FUNCTION_BLOCK ForceLimiterFSM IMPLEMENTS i_actionHandler
VAR_INPUT
	xEnable				: BOOL;				// Enable inputs and FSM operation
	MaxSnub				: LREAL; 			// Max Sbub (in negative lbs)
	MaxPull				: LREAL;			// Max Pull (lbs)
	Rih					: BOOL;				// Run in hole
	Pooh				: BOOL;				// Pull out of hole
	CriticalWeightRih	: LREAL;			// RIH critical weight (Cerburus Catastrophic Buckling, in negative lbs)
	CriticalWeightPooh	: LREAL;			// POOH critical weight ( Cerburus 80% pipe yield force, lbs)	
	SurpassTimeout 		: TIME  := T#10S;	// Limit surpass timeout value input
	SurpassThreshhold	: LREAL := 3.0;		// Limit surpass threshhod in %	
	CerberusDataLoaded 	: BOOL;				// Cerberus data loaded
	SurfaceWeight		: LREAL;			// Actual surface weight (lbs)	
END_VAR
VAR_OUTPUT
	Warn		: BOOL;	// Approaching limits warn
	CritAlarm	: BOOL;	// Limits surpassed alarm	
	ReduceForce	: BOOL;	// Fast stop while POOH, or run at slow speed while RIH
	AutoDisable	: BOOL;	// Disable automation if surface weight exceed surpass limits
	FsmError	: BOOL; // Fsm Error (TRUE when FSM errors)
END_VAR
VAR
	(* Calcution mode *)
	m_Pull			: BOOL; 	// Pull caluculation mode, weight is positive
	m_SurfaceWeight : LREAL;	// Normalized surface weight
	m_SurpassLimit	: LREAL;	// Surpassed limit
	m_Limit			: LREAL;	// Limit
	m_ApproachLimit : LREAL;	// Approaching limit
	

	(* Event Triggers *)	
	m_EnableTrigger				: R_TRIG;	// Enable event trigger
	m_LimitNotSetTrigger		: R_TRIG;	// Manual limit not set trigger
	m_LinitSetTrigger			: R_TRIG;	// Manual limit set trigger
	m_ApproachLimitTrigger		: R_TRIG;	// Approaching limit trigger
	m_NotApproachLimitTrigger	: R_TRIG; 	// Not appraching limit trigger
	m_LimitSurpassedTrigger		: R_TRIG;	// Limits surpassed trigger
	m_LimitNotSurpassedTrigger	: R_TRIG;	// Limits not surpassed trigger		
	m_SurpassTimer				: TON;		// Limit surpass timer used to detect timeout error


	(* Finite State Machine *)
	m_ForceLimiterFsmTable	: ARRAY[0..FSM_STATE_ARRAY_MAX, 0..FSM_EVENT_ARRAY_MAX, 0..FSM_ACTIONS_ARRAY_MAX] OF BYTE := [
	(* FsmState_Error --------------------------------------------------------- *)
	(*  Next State							Action								*)
	
		(* FsmEvent_Manual_Limits_Not_Set *)
		FSM_EVENT_INVALID,					ForceLimiterFsmAction.FsmAction_None,
		
		(* FsmEvent_Manual_Limits_Set *)
		FSM_EVENT_INVALID,					ForceLimiterFsmAction.FsmAction_None,
		
		(* FsmEvent_Approaching_Limits *)
		FSM_EVENT_INVALID,					ForceLimiterFsmAction.FsmAction_None,
		
		(* FsmEvent_Not_Approaching_Limits *)
		FSM_EVENT_INVALID,					ForceLimiterFsmAction.FsmAction_None,
		
		(* FsmEvent_Limit_Surpassed *)
		FSM_EVENT_INVALID,					ForceLimiterFsmAction.FsmAction_None,
		
		(* FsmEvent_Limit_Not_Surpassed *)
		FSM_EVENT_INVALID,					ForceLimiterFsmAction.FsmAction_None,	

	(* FsmState_Off ----------------------------------------------------------- *)
	(*  Next State							Action								*)
	
		(* FsmEvent_Manual_Limits_Not_Set *)
		ForceLimiterFsmState.FsmState_Off,	ForceLimiterFsmAction.FsmAction_Crit_Alarm,
		
		(* FsmEvent_Manual_Limits_Set *)
		ForceLimiterFsmState.FsmState_On,	ForceLimiterFsmAction.FsmAction_None,
		
		(* FsmEvent_Approaching_Limits *)
		ForceLimiterFsmState.FsmState_Off,	ForceLimiterFsmAction.FsmAction_None,
		
		(* FsmEvent_Not_Approaching_Limits *)
		ForceLimiterFsmState.FsmState_Off,	ForceLimiterFsmAction.FsmAction_None,
		
		(* FsmEvent_Limit_Surpassed *)
		ForceLimiterFsmState.FsmState_Off,	ForceLimiterFsmAction.FsmAction_None,
		
		(* FsmEvent_Limit_Not_Surpassed *)
		ForceLimiterFsmState.FsmState_Off,	ForceLimiterFsmAction.FsmAction_None,

	(* FsmState_On ------------------------------------------------------------ *)
	(*  Next State							Action								*)
	
		(* FsmEvent_Manual_Limits_Not_Set *)
		ForceLimiterFsmState.FsmState_Off,	ForceLimiterFsmAction.FsmAction_None,
		
		(* FsmEvent_Manual_Limits_Set *)
		ForceLimiterFsmState.FsmState_On,	ForceLimiterFsmAction.FsmAction_None,
		
		(* FsmEvent_Approaching_Limits *)
		ForceLimiterFsmState.FsmState_On,	ForceLimiterFsmAction.FsmAction_Warn,
		
		(* FsmEvent_Not_Approaching_Limits *)
		ForceLimiterFsmState.FsmState_On,	ForceLimiterFsmAction.FsmAction_Clear_Warning,
		
		(* FsmEvent_Limit_Surpassed *)
		ForceLimiterFsmState.FsmState_On,	ForceLimiterFsmAction.FsmAction_Crit_Alarm,
		
		(* FsmEvent_Limit_Not_Surpassed *)
		ForceLimiterFsmState.FsmState_On,	ForceLimiterFsmAction.FsmAction_Clear_Crit_Alarm	
	];

	m_ForceLimiterFSM : fb_FSM(	fsmId			:= ADR(	m_ForcelimiterFSM ),
								stateTable		:= ADR( m_ForceLimiterFsmTable ),
								actionHandler	:= THIS^,
								numStates		:= ForcelimiterFsmState.NUM_FsmStates,
								numEvents		:= ForceLimiterFsmEvent.NUM_FsmEvents,
								initialState	:= ForcelimiterFsmState.FsmState_Off);
								
	m_FsmError			: BOOL;					// FSM error bit (TRUE - FSM Halted)
	m_FsmErrorNum		: TFsmError;			// FSM error ENUM number
	m_FsmCurrentState	: ForceLimiterFsmState;	// Current FSM state output
	m_FsmLastState		: ForceLimiterFsmState; // Previous state used for debugging FSM errors
	m_FsmLastEvent		: ForceLimiterFsmEvent; // Last triggered event output
	m_FsmLastAction		: ForceLimiterFsmAction;// Last run action output	
END_VAR
VAR CONSTANT
	FSM_NUM_EVENT_ACTIONS	: INT := 1;
	FSM_NUM_STATES			: INT := ForceLimiterFsmState.NUM_FsmStates;
	FSM_NUM_EVENTS			: INT := ForceLimiterFsmEvent.NUM_FsmEvents;
	FSM_STATE_ARRAY_MAX		: INT := FSM_NUM_STATES - 1;
	FSM_EVENT_ARRAY_MAX		: INT := FSM_NUM_EVENTS - 1;
	FSM_ACTIONS_ARRAY_MAX	: INT := FSM_NUM_EVENT_ACTIONS;
END_VAR

// (* FSM *)

m_ForceLimiterFSM( xEnable := xEnable, xError => m_FsmError, errorNum => m_FsmErrorNum);
FsmError := m_FsmError;

m_FsmCurrentState := m_ForceLimiterFSM.FSM_GetCurrentState();

IF Pooh = TRUE AND Rih = FALSE THEN
	m_Pull := TRUE;
ELSIF Pooh = FALSE AND Rih = TRUE THEN
	m_Pull := FALSE;
END_IF

// Pull operation 
IF m_Pull = TRUE THEN

	m_SurfaceWeight := SurfaceWeight;	
	IF CerberusDataLoaded = TRUE THEN
		m_Limit	:= MIN(MaxPull, CriticalWeightPooh);		
	ELSE 
		m_Limit	:= MaxPull;		
	END_IF	

// Snub operation	
ELSE
	
	m_SurfaceWeight := -1.0* SurfaceWeight;
	IF CerberusDataLoaded = TRUE THEN
		m_Limit	:= -1.0 * MAX(MaxSnub, CriticalWeightRih);		
	ELSE 
		m_Limit	:= -1.0 * MaxSnub;		
	END_IF	
	
END_IF

m_SurpassLimit 	:= m_Limit * ( 1 + SurpassThreshhold / 100.0);		
m_ApproachLimit := m_Limit * ( 1 - SurpassThreshhold / 100.0);	

// Timing if the surface weight is larger than the limit
m_SurpassTimer(IN := (m_SurfaceWeight > m_Limit), PT := SurpassTimeout);


// (* EVENT TRIGGER *)

// Reset FSM to initialization state
m_EnableTrigger(CLK := xEnable);
IF (m_EnableTrigger.Q) THEN
	m_ForceLimiterFSM.FSM_Reset();
END_IF

// Manual limits not set
m_LimitNotSetTrigger(CLK := MaxSnub >= 0.0 OR MaxPull <= 0.0); 
IF m_LimitNotSetTrigger.Q THEN
	m_ForceLimiterFSM.FSM_ProcessEvent(ForceLimiterFsmEvent.FsmEvent_Manual_Limits_Not_Set);
END_IF

// Manual limits set
m_LinitSetTrigger(CLK := MaxSnub < 0.0 AND MaxPull > 0.0);
IF m_LinitSetTrigger.Q THEN
	m_ForceLimiterFSM.FSM_ProcessEvent(ForceLimiterFsmEvent.FsmEvent_Manual_Limits_Set);
END_IF

// Approaching the limit
m_ApproachLimitTrigger(CLK := m_SurfaceWeight >= m_ApproachLimit);
IF m_ApproachLimitTrigger.Q THEN
	m_ForceLimiterFSM.FSM_ProcessEvent(ForceLimiterFsmEvent.FsmEvent_Approaching_Limits);
END_IF

// Not approaching the limit
m_NotApproachLimitTrigger(CLK := m_SurfaceWeight < m_ApproachLimit);
IF m_NotApproachLimitTrigger.Q THEN
	m_ForceLimiterFSM.FSM_ProcessEvent(ForceLimiterFsmEvent.FsmEvent_Not_Approaching_Limits);
END_IF

// Surpassed the limit
m_LimitSurpassedTrigger(CLK := m_SurfaceWeight >= m_SurpassLimit OR m_SurpassTimer.Q);
IF m_LimitSurpassedTrigger.Q THEN
	m_ForceLimiterFSM.FSM_ProcessEvent(ForceLimiterFsmEvent.FsmEvent_Limit_Surpassed);
END_IF

// // Limit not Surpassed
m_LimitNotSurpassedTrigger(CLK := m_SurfaceWeight < m_SurpassLimit AND NOT m_SurpassTimer.Q);
IF m_LimitNotSurpassedTrigger.Q THEN
	m_ForceLimiterFSM.FSM_ProcessEvent(ForceLimiterFsmEvent.FsmEvent_Limit_Not_Surpassed);
END_IF

METHOD ExecuteAction : BOOL
VAR_INPUT
	p_FSM			: POINTER TO fb_FSM;	// Pointer to the instatiation of the FSM object
	currentAction	: TFsmAction;			// Current FSM action being processed
	currentEvent	: TFsmEventDesc;		// Current FSM event being processed
END_VAR
CASE CurrentAction OF
	
	ForceLimiterFsmAction.FsmAction_None:	
		// Return TRUE
		ExecuteAction := TRUE;
		
	ForceLimiterFsmAction.FsmAction_Warn:	
		// Generate warn, reduce speed
		Warn		:= TRUE;		
		ReduceForce	:= TRUE;		
		
		// Return TRUE
		ExecuteAction := TRUE;
	
	ForceLimiterFsmAction.FsmAction_Crit_Alarm:
		// Generate critical alarm, disable cruise control and auto mill
		CritAlarm	:= TRUE;		
		AutoDisable	:= TRUE;		

		// Return TRUE
		ExecuteAction := TRUE;		
	
	ForceLimiterFsmAction.FsmAction_Clear_Warning:
		// Clear warning, reduce speed
		Warn		:= FALSE;		
		ReduceForce	:= FALSE;

		// Return TRUE
		ExecuteAction := TRUE;		
		
	ForceLimiterFsmAction.FsmAction_Clear_Crit_Alarm:
		// Clear critical alarm, enable cruise control and auto mill
		CritAlarm	:= FALSE;		
		AutoDisable	:= FALSE;		

		// Return TRUE
		ExecuteAction := TRUE;		
	
	FSM_ACTION_UNEXPECTED_EVENT:
		// Do action unexpected event
		p_FSM^.FSM_ASSERT(FALSE, TFsmError.FSM_INVALID_ACTION);
		
		// Return FALSE
		ExecuteAction := FALSE;
		
	FSM_ACTION_ERROR_EVENT:
		// Do action error event
		m_EnableTrigger(CLK := FALSE);
		
		// Return FALSE
		ExecuteAction := FALSE;

ELSE
	// Error trap - Unknow action
	p_FSM^.FSM_ASSERT(FALSE, TFsmError.FSM_INVALID_ACTION);
	
	// Return FALSE
	ExecuteAction := FALSE;

END_CASE

m_FsmLastState	:= p_FSM^.FSM_GetPreviousState();
m_FsmLastEvent	:= currentEvent.event;
m_FsmLastAction	:= currentAction;
END_METHOD

END_FUNCTION_BLOCK

(* stored: Version 1.1.0.1, ProductVersion 3.1.4024.6
   POU ForceLimiterFSM: Id {343a6fe0-52b1-49d8-9ae1-c1152df0e24c}, SpecialFunc None
   Method ExecuteAction: Id {065d9514-3328-412e-967a-dbc899eb9f38} *)
